FUNCTION_BLOCK SCREW_STATION_MANAGER
  {SET_ATTRIBUTE(OpcUa, SERVICE)}
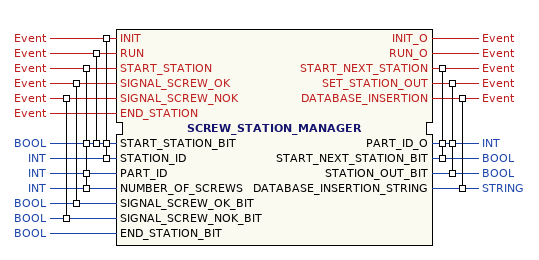
  EVENT_INPUT
    INIT WITH STATION_ID, START_STATION_BIT;
    RUN WITH START_STATION_BIT;
    START_STATION WITH START_STATION_BIT, PART_ID, NUMBER_OF_SCREWS;
    SIGNAL_SCREW_OK WITH SIGNAL_SCREW_OK_BIT;
    SIGNAL_SCREW_NOK WITH SIGNAL_SCREW_NOK_BIT;
    END_STATION;
  END_EVENT
  EVENT_OUTPUT
    INIT_O;
    RUN_O;
    START_NEXT_STATION WITH PART_ID_O, START_NEXT_STATION_BIT;
    SET_STATION_OUT WITH STATION_OUT_BIT, PART_ID_O;
    DATABASE_INSERTION WITH DATABASE_INSERTION_STRING;
  END_EVENT
  VAR_INPUT
    START_STATION_BIT : BOOL;
    STATION_ID : INT;
    PART_ID : INT;
    NUMBER_OF_SCREWS : INT;
    SIGNAL_SCREW_OK_BIT : BOOL;
    SIGNAL_SCREW_NOK_BIT : BOOL;
    END_STATION_BIT : BOOL;
  END_VAR
  VAR_OUTPUT
    PART_ID_O : INT; {SET_ATTRIBUTE(OpcUa, Variable.RUN)}
    START_NEXT_STATION_BIT : BOOL; {SET_ATTRIBUTE(OpcUa, Variable.RUN)}
    STATION_OUT_BIT : BOOL; {SET_ATTRIBUTE(OpcUa, Variable.RUN)}
    DATABASE_INSERTION_STRING : STRING; {SET_ATTRIBUTE(OpcUa, Variable.RUN)}
  END_VAR
END_FUNCTION_BLOCK
